(* CoDeSys 2.3 export: F_WRITE_SE_CYLINDER_POS_CFG.EXP *)

(* POU FUN/PARAMETERS/F_WRITE_SE_CYLINDER_POS_CFG, ST *)
FUNCTION F_WRITE_SE_CYLINDER_POS_CFG : BOOL
VAR_INPUT
	sHead : STRING;
	wSize   :DWORD;
	pBuffer :POINTER TO BYTE;
END_VAR
VAR_IN_OUT
	wPos     : DWORD;
	stConfig : ST_SE_CYLINDER_POS_CFG;
END_VAR
VAR
END_VAR
F_ADD_STRINGX3_TO_BUFFER( S1:= '$n#', S2:= sHead, S3:=' - Parameters:$n', wSize := wSize, pBuffer := pBuffer, wPos := wPos );

F_ADD_STRINGX4_TO_BUFFER( S1:= CONCAT(sHead, '_Ease'    ), S2:='$t', S3:= REAL_TO_STRING( stConfig.Ease    ), S4:='$n', wSize := wSize, pBuffer := pBuffer, wPos := wPos );

F_ADD_STRINGX4_TO_BUFFER( S1:= CONCAT(sHead, '_TgtLS_In'  ), S2:='$t', S3:= REAL_TO_STRING( stConfig.TgtLS_In  ), S4:='$n', wSize := wSize, pBuffer := pBuffer, wPos := wPos );
F_ADD_STRINGX4_TO_BUFFER( S1:= CONCAT(sHead, '_TgtLS_Out' ), S2:='$t', S3:= REAL_TO_STRING( stConfig.TgtLS_Out ), S4:='$n', wSize := wSize, pBuffer := pBuffer, wPos := wPos );
F_ADD_STRINGX4_TO_BUFFER( S1:= CONCAT(sHead, '_TgtLS_Slow' ), S2:='$t', S3:= REAL_TO_STRING( stConfig.TgtLS_Slow ), S4:='$n', wSize := wSize, pBuffer := pBuffer, wPos := wPos );

F_ADD_STRINGX4_TO_BUFFER( S1:= CONCAT(sHead, '_TimeMax'  ), S2:='$t', S3:= REAL_TO_STRING( stConfig.TimeMax  ), S4:='$n', wSize := wSize, pBuffer := pBuffer, wPos := wPos );
F_ADD_STRINGX4_TO_BUFFER( S1:= CONCAT(sHead, '_TimeEase' ), S2:='$t', S3:= REAL_TO_STRING( stConfig.TimeEase ), S4:='$n', wSize := wSize, pBuffer := pBuffer, wPos := wPos );

F_ADD_STRINGX4_TO_BUFFER( S1:= CONCAT(sHead, '_LS_Limit_In'  ), S2:='$t', S3:= BOOL_TO_STRING( stConfig.LS_Limit_In  ), S4:='$n', wSize := wSize, pBuffer := pBuffer, wPos := wPos );
F_ADD_STRINGX4_TO_BUFFER( S1:= CONCAT(sHead, '_LS_Limit_Out' ), S2:='$t', S3:= BOOL_TO_STRING( stConfig.LS_Limit_Out ), S4:='$n', wSize := wSize, pBuffer := pBuffer, wPos := wPos );

F_ADD_STRINGX4_TO_BUFFER( S1:= CONCAT(sHead, '_HP'  ), S2:='$t', S3:= BYTE_TO_STRING( stConfig.HP ), S4:='$n', wSize := wSize, pBuffer := pBuffer, wPos := wPos );
END_FUNCTION
